// TIA Portal V17 export
// export: Created 2024-06-14T09:53:05.3245941Z, ExportSetting WithDefaults, DisplayName Totally Integrated Automation Portal, DisplayVersion V17, DisplayName TIA Portal Openness, DisplayVersion V17, DisplayName TIA Portal Version Control Interface, DisplayVersion V17, DisplayName Simotion SCOUT TIA, DisplayVersion 5.4.3.0, DisplayName SINAMICS Startdrive Advanced, DisplayVersion V17 SP1 Update 1, DisplayName SINAMICS Startdrive G110M, G120, G120C, G120D, G120P, G115D, DisplayVersion V17 SP1 Update 1, DisplayName SINAMICS Startdrive G130, G150, S120, S150, SINAMICS MV, S210, DisplayVersion V17 SP1 Update 1, DisplayName STEP 7 Professional, DisplayVersion V17, DisplayName STEP 7 Safety, DisplayVersion V17, DisplayName WinCC Professional, DisplayVersion V17
DATA_BLOCK "L2_Total Enabled Station_DB"   // DB19
VERSION : 0.1
// stored: AutoNumber true, DBAccessibleFromOPCUA true, InstanceOfName Total Enabled Station, InstanceOfType FB
"Total Enabled Station"
   // VAR_INPUT
   //    Enable_Station1 : Bool;
   //    Enable_Station4 : Bool;
   //    Enable_Station5 : Bool;
   //    S1_Enabled_Station : Array[1..6] of Bool;
   //    S4_Enabled_Station : Array[1..6] of Bool;
   //    S5_Enabled_Station : Array[1..6] of Bool;
   // END_VAR
   // VAR_OUTPUT
   //    Enabled_Station_S1 : Int;
   //    Enabled_Station_S4 : Int;
   //    Enabled_Station_S5 : Int;
   // END_VAR
   // VAR
   //    Enabled_Station1 { S7_SetPoint := 'True'} : "Enabled_Station";
   //    Enabled_Station4 { S7_SetPoint := 'True'} : "Enabled_Station";
   //    Enabled_Station5 { S7_SetPoint := 'True'} : "Enabled_Station";
   // END_VAR
BEGIN
END_DATA_BLOCK
